(* CoDeSys 2.3.9.37 project: Cap8_2.pro *)
(* Libraries: Standard.lib 4.10.05 12:14:46 *)

(* Global variable list: Global_Variables *)
VAR_GLOBAL
       (* Entradas *)
	Interruptor: BOOL;
       (* Salida *)
	Luz: BOOL;
END_VAR

(* POU PLC_PRG, LD *)
PROGRAM PLC_PRG
VAR

END_VAR
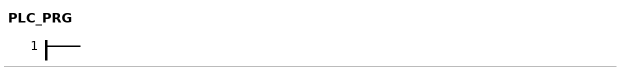
_LD_ (* Ladder Diagram *)
NETWORK 1
	*
_END_LD_
(* the same logic as Structured Text *)
(* Network 1 *)
END_PROGRAM

(* Visualisation Visu
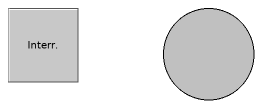
button at (60,89)-(130,163): text "Interr."; toggles Interruptor
ellipse at (215,89)-(306,181): alarm colour if Luz
*)
